FUNCTION_BLOCK SF_EmergencyStop (* PLCopen Safety SF_EmergencyStop (Part 1 v2.10, Ch. 6.5) - Emergency Stop Monitoring *)
  (* Standard: 61499-2; Function: Monitors an emergency stop sensor (S_EStopIn). S_EStopOut only returns TRUE after S_EStopIn is TRUE again AND an acknowledgment (S_StartReset/S_AutoReset/Reset) occurred, per EN ISO 13849-1:2015 5.2.2 / IEC 60204-1:2016 9.2.3.4.; Description: Copyright (c) 2026 Meisterschulen am Ostbahnhof This program and the accompanying materials are made available under the terms of the Eclipse Public License 2.0 which is available at https://www.eclipse.org/legal/epl-2.0/ SPDX-License-Identifier: EPL-2.0 *)
  (* Version 1.1, 2026-10-09, Franz Höpfinger, Meisterschulen am Ostbahnhof, Added EReset event input (REQ[...] Reset-edge checks replaced by EReset[...], xPrevReset removed). Non-literal 61499 extension, pairs with SF_ResetButton.EResetOut: no external gate FB needed any more to synthesize the reset-edge event. *)
  (* Version 1.0, 2026-10-09, Franz Höpfinger, Meisterschulen am Ostbahnhof, ECC reconstructed from PLCopen Safety Part 1 v2.10 Ch. 6.5.3 (Functional Description) and Ch. 6.5.6 (DiagCode table), not from Figure 23 directly (OCR of that state diagram was unreliable, same issue previously found and corrected in SF_ResetButton/Figure 15). Verify against the real Figure 23 image if available. Source: PLCopen TC5 Safety Part 1, Version 2.10, Nov. 7 2023, Chapter 6.5 Emergency Stop Function. *)
  PACKAGE logiBUS::safety::PLCopen;
  IMPORT logiBUS::safety::PLCopen::const::DiagCodes;
  IMPORT logiBUS::safety::PLCopen::const::EmergencyStopDiagCodes;
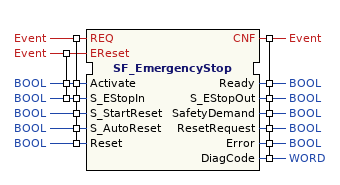
  EVENT_INPUT
    REQ WITH Activate, S_EStopIn, S_StartReset, S_AutoReset, Reset; (* Cyclic evaluation request *)
    EReset WITH Activate, S_EStopIn; (* Dedicated reset-edge event, in addition to REQ. Typically fed directly by SF_ResetButton.EResetOut *)
  END_EVENT
  EVENT_OUTPUT
    CNF WITH Ready, S_EStopOut, SafetyDemand, ResetRequest, Error, DiagCode; (* Confirmation of Requested Service *)
  END_EVENT
  VAR_INPUT
    Activate : BOOL := FALSE; (* FB enable. FALSE=inactive (sIdle) *)
    S_EStopIn : BOOL := FALSE; (* Emergency stop sensor. FALSE=stop engaged (demand), TRUE=not engaged *)
    S_StartReset : BOOL := FALSE; (* TRUE=auto-acknowledge the first time this FB is activated *)
    S_AutoReset : BOOL := FALSE; (* TRUE=auto-acknowledge every later S_EStopIn recovery, no Reset needed *)
    Reset : BOOL := FALSE; (* Manual reset. Typically fed by the paired SF_ResetButton.ResetOut *)
  END_VAR
  VAR_OUTPUT
    Ready : BOOL := FALSE; (* FB active, outputs valid *)
    S_EStopOut : BOOL := FALSE; (* TRUE=no demand, acknowledged, safe to run *)
    SafetyDemand : BOOL := FALSE; (* TRUE while waiting for S_EStopIn to recover *)
    ResetRequest : BOOL := FALSE; (* Feeds the paired SF_ResetButton.ResetRequested input *)
    Error : BOOL := FALSE; (* TRUE while in an error state, see DiagCode *)
    DiagCode : WORD := 16#0000; (* FB-specific status/error code, see PLCopen Safety Part 1 Ch. 6.5.6 *)
  END_VAR
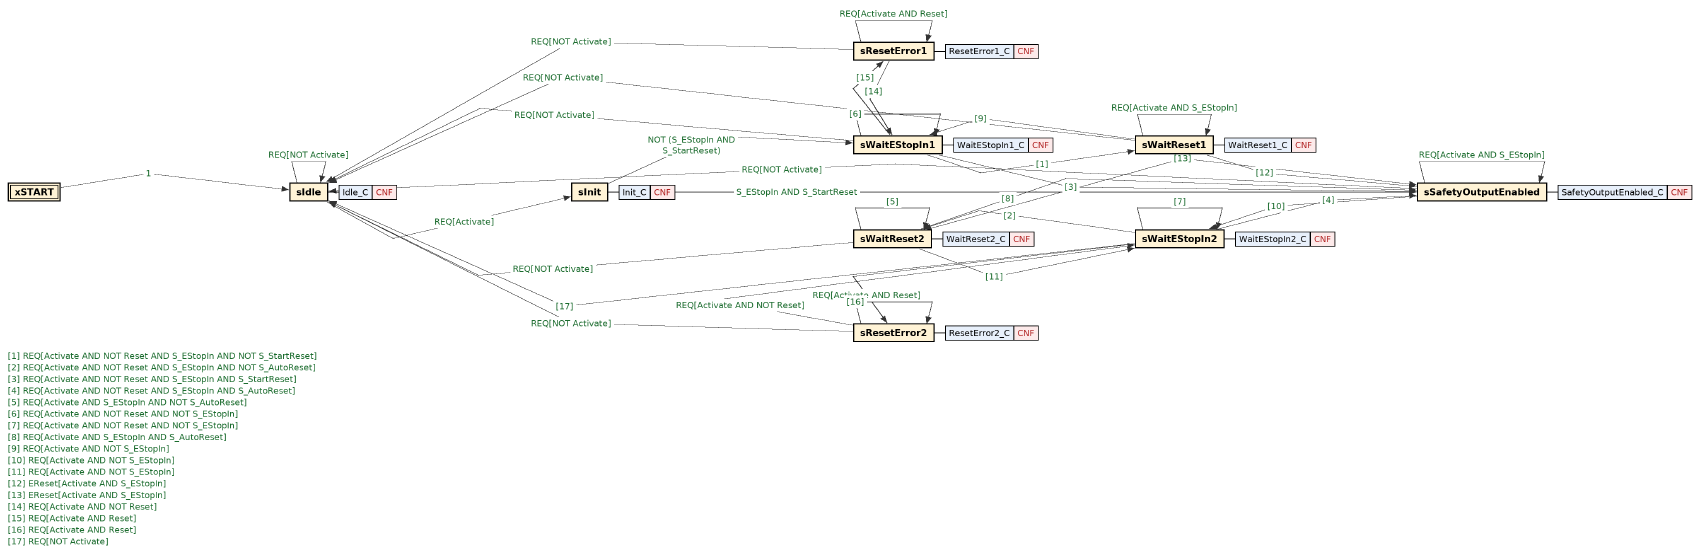
  EC_STATES
    xSTART; (* Initial State *)
    sIdle : Idle_C -> CNF;
    sInit : Init_C -> CNF; (* One-shot: branch on S_EStopIn/S_StartReset, then fall through *)
    sWaitEStopIn1 : WaitEStopIn1_C -> CNF; (* First activation: waiting for S_EStopIn *)
    sResetError1 : ResetError1_C -> CNF;
    sWaitReset1 : WaitReset1_C -> CNF; (* First activation: waiting for a rising edge on Reset *)
    sSafetyOutputEnabled : SafetyOutputEnabled_C -> CNF;
    sWaitEStopIn2 : WaitEStopIn2_C -> CNF; (* Subsequent cycles: waiting for S_EStopIn *)
    sResetError2 : ResetError2_C -> CNF;
    sWaitReset2 : WaitReset2_C -> CNF; (* Subsequent cycles: waiting for S_AutoReset or a Reset edge *)
  END_STATES
  EC_TRANSITIONS
    xSTART TO sIdle := 1;
    sIdle TO sIdle := REQ[NOT Activate];
    sIdle TO sInit := REQ[Activate];
    sInit TO sSafetyOutputEnabled := S_EStopIn AND S_StartReset;
    sInit TO sWaitEStopIn1 := NOT (S_EStopIn AND S_StartReset);
    sWaitEStopIn1 TO sIdle := REQ[NOT Activate];
    sWaitEStopIn1 TO sResetError1 := REQ[Activate AND Reset];
    sWaitEStopIn1 TO sSafetyOutputEnabled := REQ[Activate AND NOT Reset AND S_EStopIn AND S_StartReset];
    sWaitEStopIn1 TO sWaitReset1 := REQ[Activate AND NOT Reset AND S_EStopIn AND NOT S_StartReset];
    sWaitEStopIn1 TO sWaitEStopIn1 := REQ[Activate AND NOT Reset AND NOT S_EStopIn];
    sResetError1 TO sIdle := REQ[NOT Activate];
    sResetError1 TO sResetError1 := REQ[Activate AND Reset];
    sResetError1 TO sWaitEStopIn1 := REQ[Activate AND NOT Reset];
    sWaitReset1 TO sIdle := REQ[NOT Activate];
    sWaitReset1 TO sWaitEStopIn1 := REQ[Activate AND NOT S_EStopIn];
    sWaitReset1 TO sWaitReset1 := REQ[Activate AND S_EStopIn];
    sWaitReset1 TO sSafetyOutputEnabled := EReset[Activate AND S_EStopIn];
    sSafetyOutputEnabled TO sIdle := REQ[NOT Activate];
    sSafetyOutputEnabled TO sWaitEStopIn2 := REQ[Activate AND NOT S_EStopIn];
    sSafetyOutputEnabled TO sSafetyOutputEnabled := REQ[Activate AND S_EStopIn];
    sWaitEStopIn2 TO sIdle := REQ[NOT Activate];
    sWaitEStopIn2 TO sResetError2 := REQ[Activate AND Reset];
    sWaitEStopIn2 TO sSafetyOutputEnabled := REQ[Activate AND NOT Reset AND S_EStopIn AND S_AutoReset];
    sWaitEStopIn2 TO sWaitReset2 := REQ[Activate AND NOT Reset AND S_EStopIn AND NOT S_AutoReset];
    sWaitEStopIn2 TO sWaitEStopIn2 := REQ[Activate AND NOT Reset AND NOT S_EStopIn];
    sResetError2 TO sIdle := REQ[NOT Activate];
    sResetError2 TO sResetError2 := REQ[Activate AND Reset];
    sResetError2 TO sWaitEStopIn2 := REQ[Activate AND NOT Reset];
    sWaitReset2 TO sIdle := REQ[NOT Activate];
    sWaitReset2 TO sWaitEStopIn2 := REQ[Activate AND NOT S_EStopIn];
    sWaitReset2 TO sSafetyOutputEnabled := REQ[Activate AND S_EStopIn AND S_AutoReset];
    sWaitReset2 TO sWaitReset2 := REQ[Activate AND S_EStopIn AND NOT S_AutoReset];
    sWaitReset2 TO sSafetyOutputEnabled := EReset[Activate AND S_EStopIn];
  END_TRANSITIONS
  ALGORITHM Idle_C IN ST:
 // 0000 Idle - FB not active
Ready := BOOL#FALSE;
S_EStopOut := BOOL#FALSE;
SafetyDemand := BOOL#FALSE;
ResetRequest := BOOL#FALSE;
Error := BOOL#FALSE;
DiagCode := DiagCodes::IDLE;
  END_ALGORITHM
  ALGORITHM Init_C IN ST:
 // 8001 Init - activated, checking S_StartReset
Ready := BOOL#TRUE;
S_EStopOut := BOOL#FALSE;
SafetyDemand := BOOL#FALSE;
ResetRequest := BOOL#FALSE;
Error := BOOL#FALSE;
DiagCode := EmergencyStopDiagCodes::INIT;
  END_ALGORITHM
  ALGORITHM WaitEStopIn1_C IN ST:
 // 8802 Wait for S_EStopIn 1 - first activation, waiting for S_EStopIn
Ready := BOOL#TRUE;
S_EStopOut := BOOL#FALSE;
SafetyDemand := BOOL#TRUE;
ResetRequest := BOOL#FALSE;
Error := BOOL#FALSE;
DiagCode := EmergencyStopDiagCodes::WAIT_ESTOP_IN_1;
  END_ALGORITHM
  ALGORITHM ResetError1_C IN ST:
 // C001 Reset Error 1 - Reset stuck TRUE while waiting for S_EStopIn
Ready := BOOL#TRUE;
S_EStopOut := BOOL#FALSE;
SafetyDemand := BOOL#FALSE;
ResetRequest := BOOL#FALSE;
Error := BOOL#TRUE;
DiagCode := EmergencyStopDiagCodes::RESET_ERROR_1;
  END_ALGORITHM
  ALGORITHM WaitReset1_C IN ST:
 // 8402 Wait for Reset 1 - S_EStopIn is TRUE, waiting for a rising edge on Reset
Ready := BOOL#TRUE;
S_EStopOut := BOOL#FALSE;
SafetyDemand := BOOL#FALSE;
ResetRequest := BOOL#TRUE;
Error := BOOL#FALSE;
DiagCode := EmergencyStopDiagCodes::WAIT_RESET_1;
  END_ALGORITHM
  ALGORITHM SafetyOutputEnabled_C IN ST:
 // 8000 Safety Output Enabled
Ready := BOOL#TRUE;
S_EStopOut := BOOL#TRUE;
SafetyDemand := BOOL#FALSE;
ResetRequest := BOOL#FALSE;
Error := BOOL#FALSE;
DiagCode := EmergencyStopDiagCodes::SAFETY_OUTPUT_ENABLED;
  END_ALGORITHM
  ALGORITHM WaitEStopIn2_C IN ST:
 // 8804 Wait for S_EStopIn 2 - safety demand detected, waiting for S_EStopIn
Ready := BOOL#TRUE;
S_EStopOut := BOOL#FALSE;
SafetyDemand := BOOL#TRUE;
ResetRequest := NOT Reset;
Error := BOOL#FALSE;
DiagCode := EmergencyStopDiagCodes::WAIT_ESTOP_IN_2;
  END_ALGORITHM
  ALGORITHM ResetError2_C IN ST:
 // C011 Reset Error 2 - Reset stuck TRUE while waiting for S_EStopIn
Ready := BOOL#TRUE;
S_EStopOut := BOOL#FALSE;
SafetyDemand := BOOL#FALSE;
ResetRequest := BOOL#FALSE;
Error := BOOL#TRUE;
DiagCode := EmergencyStopDiagCodes::RESET_ERROR_2;
  END_ALGORITHM
  ALGORITHM WaitReset2_C IN ST:
 // 8404 Wait for Reset 2 - waiting for S_AutoReset or a rising edge on Reset
Ready := BOOL#TRUE;
S_EStopOut := BOOL#FALSE;
SafetyDemand := BOOL#FALSE;
ResetRequest := NOT Reset;
Error := BOOL#FALSE;
DiagCode := EmergencyStopDiagCodes::WAIT_RESET_2;
  END_ALGORITHM
END_FUNCTION_BLOCK
(* other elements stored in the file *)
(* 6.5.3: S_StartReset only matters on this very first activation. If S_EStopIn is already TRUE and S_StartReset is set, go straight to Enabled; otherwise wait. *)
